// TIA Portal V21 export
FUNCTION_BLOCK "AxisAS_Mng"   // FB81, LAD
TITLE = Positioner + PID / Controllo asse + PID
{ S7_Optimized_Access := 'TRUE' }
VERSION : 1.0
// Positioner with Pid management
// 
// Version from master S7: 2.6
// 
// Date: 2017-08-25
// Project: Mora A.
// 
// Version 2.7: -Corrected maximum speed reached in proportional calculation check.
// Version 2.8: -Used Type for CFG data.
// Gestore ASSE per motore asincrono con posizionatore a generazione di profilo ed inseguimento proporzionale + piramidale
// 
// Michele Montanari
// 
// ver 0.0
// - Curva Trapezio
// - Curva "esse" logaritmica
// - Auto gestione curva per piccoli spostamenti
// - Attesa segnale inverter magnetizzato
// 
// ver 1.0 24/01/2023
// - Curva "esse" Coseno
// - Aggiornamneto struttura
// - Calcolo di tutte le curve in simultanea
// - Arresto #Out in posizione su finestra Vir (da provare.... anche su velocità  == 0)
// - Autogestione (selezione) calcolo acc e dec su definizione prestazioni massime
// - Autogestione (selezione) calcolo velocità possibile in funzione del nuovo target
// - Richiesta abilitazione inverter sempre attiva per abbattere tempo di magentizzazione
// - Inversione al volo del moto
// - Gestione interna del freno motore
// stored: MemoryReserve 100, SetENOAutomatically false
   VAR RETAIN
      DataIn : Struct   // Comando asse
         ixEnablePos { S7_SetPoint := 'True'} : Bool;   // Enable positioner / Abilita asse
         ixDriveReady { S7_SetPoint := 'True'} : Bool;   // Inverter magnetizzato
         ixEnableLevRes { S7_SetPoint := 'True'} : Bool;   // Enable level research / Abilita ricerca livello
         ixAlarmReset { S7_SetPoint := 'True'} : Bool;   // Reset alarms / Reset allarmi
         ixAbort { S7_SetPoint := 'True'} : Bool;   // Initializing motor encoder position / Abort sistema
         ixJogPos { S7_SetPoint := 'True'} : Bool;   // Manual Jog positive / Manuale JOG +
         ixJogNeg { S7_SetPoint := 'True'} : Bool;   // Manual Jog negative / Manuale JOG -
         xAutoSpeedDetect { S7_SetPoint := 'True'} : Bool;   // Calcolo velocità automatico su movimento
         xAutoAccDecCalculation { S7_SetPoint := 'True'} : Bool;   // Calcolo Acc Dec automatico su velocità
         ifPositionRequest { S7_SetPoint := 'True'} : Real;   // Position requested (mm) / Quota richiesta (mm)
         ifSpeedRequest { S7_SetPoint := 'True'} : Real;   // Speed requested (mm/sec) / Velocità richiesta (mm/sec)
         ifPositionStartLev { S7_SetPoint := 'True'} : Real;   // Position start research (mm) / Quota inizio ricerca (mm)
         ifSpeedLev { S7_SetPoint := 'True'} : Real;   // Research speed (mm/sec) / Velocità ricerca (mm/sec)
         ifAccRamp { S7_SetPoint := 'True'} : Real;   // Acceleration ramp (mm/sec^2) / * Rampa accelerazione (mm/sec^2)
         ifDecRamp { S7_SetPoint := 'True'} : Real;   // Deceleration ramp (mm/sec^2) / * Rampa decelerazione (mm/sec^2)
         ifTimeScan { S7_SetPoint := 'True'} : Real;   // Time last scan (sec) / Tempo ultima scansione (sec)
         ifEncoder { S7_SetPoint := 'True'} : Real;   // Actual encoder position (encoder) / Posizione attuale encoder
      END_STRUCT;
      DataOut : Struct   // Gestione Inverte e posizioni
         oxCmdMotorForw : Bool;   // Inverter run enabled / Abilitazione marcia Avanti
         oxCmdMotorBack : Bool;   // Abilitazione marcia Indietro
         oxCmdBrake : Bool;   // Enable brake release / Comando stacco freno
         oxPosError { S7_SetPoint := 'True'} : Bool;   // Pursuit error / Allarme: Errore di inseguimento
         oxEndPos : Bool;   // Positioning terminated / Posizionamento terminato
         oxEndPosBig : Bool;   // Posizionamento Allargato terminato
         oxStopSpeed : Bool;   // Motor speed below low limit / Velocità motore = 0
         oxAccOnWork : Bool;   // Rampa Acc in atto
         oxDecOnWork : Bool;   // Rampa Dec in atto
         ofSpeedRequest : Real;   // Motor speed requested (mm/sec) / Velocita motore richiesta (mm/sec)
         ofEncMotorPos : Real;   // Motor encoder position (mm) / Posizione encoder motore (mm)
         ofMaxError : Real;   // Pursuit max error (mm) / Errore massimo di inseguimento (mm)
         ofSpaceStop : Real;   // Stop space requested from current position/speed (mm) / Spazio richiesto per fermata da posizione/velocità attuale (mm)
         ofSpaceLevRes : Real;   // Spazio richiesto per cambio velocità ricerca livello da posizione/velocità attuale (mm)
         ofSpaceStart : Real;   // Spazio richiesto per partenza da posizione/velocità attuale (mm)
         otTimeMove : Time;   // Tempo ultimo movimento
      END_STRUCT;
      Cfg { S7_SetPoint := 'True'} : "AxixAS_CFG_Type";   // Block data initialisation / Configurazione Asse
      Work : Struct   // Positioner management / Gestione Asse
         xEnablePos { S7_SetPoint := 'True'} : Bool;   // Positioner enabled / Posizionatore abilitato/Positioner enabled
         xINEnable : Bool;   // Memo Posizionatore abilitato per inversione
         xDriveReady { S7_SetPoint := 'True'} : Bool;   // Inverter magnetizzato
         xCmdVirSpeedChanged { S7_SetPoint := 'True'} : Bool;   // Variazione target VEL durante missione
         "xCurveS-L" { S7_SetPoint := 'True'} : Bool;   // Curva non lineare
         "xAutoChangeS-L" { S7_SetPoint := 'True'} : Bool;   // Autoimpostazione LIN per brevi spostamenti
         "xCTRAutoChangeS-L" { S7_SetPoint := 'True'} : Bool;   // Autoimpostazione LIN per brevi spostamenti
         xDecStop { S7_SetPoint := 'True'} : Bool;   // Start dec. for reached requested position / Inizio dec. per raggiungimento quota richiesta
         xDecResearch { S7_SetPoint := 'True'} : Bool;   // Deceleration start for moving to level search speed / Inizio decelerazione per passaggio a velocità ricerca livello
         xStopVirPositioner { S7_SetPoint := 'True'} : Bool;   // Stop positioner for pos. reached / Arresto posizionatore Target raggiunto
         xEnableJog { S7_SetPoint := 'True'} : Bool;   // Jog movement in progress / JOG movimento in corso
         f_PositionTarget { S7_SetPoint := 'True'} : Real;   // Posizione Richiesta Target
         fVirPos { S7_SetPoint := 'True'} : Real;   // Pos. virtual encoder positioner (mm) / Posizione encoder Asse virtuale (mm)
         f_SpeedReqCalc { S7_SetPoint := 'True'} : Real;   // Velocità TARGET autocalcolata su spazio destinazione
         fVirSpeed { S7_SetPoint := 'True'} : Real;   // Virtual encoder speed positioner (mm/sec) / Velocità Asse virtuale (mm/sec) TRA-LOG-COS
         fVirSpeedLinear { S7_SetPoint := 'True'} : Real;   // Velocità Asse LINEARE
         fVirSpeedLog { S7_SetPoint := 'True'} : Real;   // Velocità Asse LOGARITMICA
         fVirSpeedCos { S7_SetPoint := 'True'} : Real;   // Velocità Asse COSENO
         fCmdVirSpeed { S7_SetPoint := 'True'} : Real;   // Virtual encoder current sp(mm/sec) / Velocità richiesta Asse (mm/sec)
         fCmdVirSpeedMemo { S7_SetPoint := 'True'} : Real;   // Memo Velocità richiesta Asse (mm/sec)
         fCmdVirAcc { S7_SetPoint := 'True'} : Real;   // Acc requested for positioner (mm/sec^2) / Acc. richiesta Asse (mm/sec^2)
         fCmdVirDec { S7_SetPoint := 'True'} : Real;   // Dec. requested for positioner (mm/sec^2) / Dec. richiesta Asse (mm/sec^2)
         fLimVirDec { S7_SetPoint := 'True'} : Real;   // Max modulated dec. limit to stop / * Limite massimo dec. modulata per fermata
         fDecVirStop { S7_SetPoint := 'True'} : Real;   // Dec. requested for positioner stop height (mm/sec^2) / * Dec. richiesta per posizionatore stop quota (mm/sec^2)
         fCalcEncErr { S7_SetPoint := 'True'} : Real;   // Error between motor encoder current & real pos. (mm) / * Errore tra pos. attuale e reale encoder motore
         fJogSpeed { S7_SetPoint := 'True'} : Real;   // Speed gen. by jog movement (mm/sec) / Velocità JOG (mm/sec)
         fCmdJogSpeed { S7_SetPoint := 'True'} : Real;   // Speed request to jog movement (mm/sec) / Velocità richiesta JOG (mm/sec)
         fCmdJogAcc { S7_SetPoint := 'True'} : Real;   // Acc. requested for jog movement (mm/sec^2) / Acc. richiesta JOG (mm/sec^2)
         fCmdJogDec { S7_SetPoint := 'True'} : Real;   // Dec. requested for jog movement (mm/sec^2) / Dec. richiesta JOG (mm/sec^2)
         "fLim+Ppid" { S7_SetPoint := 'True'} : Real;   // Proportional action positive maximum limit (1/5 max speed) / Limite massimo positivo azione proporzionale (20% velocità massima)
         "fLim-Ppid" { S7_SetPoint := 'True'} : Real;   // Proportional action negative maximum limit (1/5 max speed) / Limite massimo negativo azione proporzionale (20% velocità massima)
         fCmdSpeedMot { S7_SetPoint := 'True'} : Real;   // Motor control speed from positioner o Jog / Velocità comando motore da POS o JOG
         fSuppCalcPpid { S7_SetPoint := 'True'} : Real;   // Proportional calculation supp. / App calcolo proporzionale
         fMemoMaxSpeed { S7_SetPoint := 'True'} : Real;   // Store maximum speed (mm/sec) / Memorizzo velocità massima (mm/sec)
         fPpid { S7_SetPoint := 'True'} : Real;   // Part P of Pid / Parte P del Pid
         fMemoOldPos { S7_SetPoint := 'True'} : Real;   // Quota Old/Position Old (mm)
         fAccOnWork { S7_SetPoint := 'True'} : Real;   // Accelerazione calcolata/imposta
         fDecOnWork { S7_SetPoint := 'True'} : Real;   // Decelerazione calcolata/imposta
         xTimBrakeDelay_Fwd : Bool;   // Ritardo sgancio freno FWD
         xTimBrakeDelay_Bkw : Bool;   // Ritardo sgancio freno BKW
         xTimStopEndPos : Bool;   // Ritardo allarme controllo fine posizionamento
         fCalc : Array[0..20] of Real;
         xCalc : Array[0..20] of Bool;
      END_STRUCT;
   END_VAR
   VAR
      TmrBrake_Fwd : IEC_TIMER;   // Timer sgancio freno FWD
      TmrBrake_Bkw : IEC_TIMER;   // Timer sgancio freno BKW
      Tmr_EndPos : IEC_TIMER;   // Timer allarme controllo fine posizionamento
      Tmr_DriveOnReq : IEC_TIMER;   // Timer OFF richiesta Drive Ready
      Tmr_OnMove : IEC_TIMER;
   END_VAR
   VAR_TEMP
      tfSuppCalc : Real;   // Calculation support / Appoggio per calcoli
      fSlopeAccLog : Real;
      fSlopeDecLog : Real;
      fSlopeAccCos : Real;
      fSlopeDecCos : Real;
      fCalcSpeed : Real;
      oxCmdMotorFWD : Bool;
      oxCmdMotorBKW : Bool;
      fCalcSpaceOff : Real;
      xDummy : Bool;
   END_VAR
   VAR CONSTANT
      PiGrego : Real := 3.141593;
      "100Sec" : Time := T#100s;
   END_VAR
   VAR_TEMP   // added for the SCL form of the ladder/FBD networks
      _w1 : Bool;
      _w2 : Bool;
      _w3 : Bool;
   END_VAR
BEGIN

REGION Network 1 (SCL): Autocalcolo velocità su spazio da percorrere
   IF #DataIn.xAutoSpeedDetect THEN
       IF #Cfg."xmm/degree" THEN
           IF ABS(#DataIn.ifPositionRequest - #DataIn.ifEncoder) >= #Cfg.fMaxSpeed / 2 THEN
               #Work.f_SpeedReqCalc := #DataIn.ifSpeedRequest;
           ELSE
               #fCalcSpeed := ABS(#DataIn.ifPositionRequest - #DataIn.ifEncoder);
               IF NOT #DataOut.oxCmdMotorForw AND NOT #DataOut.oxCmdMotorBack THEN
                   IF #fCalcSpeed <= #DataIn.ifSpeedRequest THEN
                       #Work.f_SpeedReqCalc := #fCalcSpeed;
                   ELSE
                       #Work.f_SpeedReqCalc := #DataIn.ifSpeedRequest;
                   END_IF;
               END_IF;
           END_IF;
       ELSE
           IF ABS(#DataIn.ifPositionRequest - #DataIn.ifEncoder) >= 60.0 THEN
               #Work.f_SpeedReqCalc := #DataIn.ifSpeedRequest;
           ELSE
               #fCalcSpeed := ABS(#DataIn.ifPositionRequest - #DataIn.ifEncoder);
               IF NOT #DataOut.oxCmdMotorForw AND NOT #DataOut.oxCmdMotorBack THEN
                   IF #fCalcSpeed <= #DataIn.ifSpeedRequest THEN
                       #Work.f_SpeedReqCalc := #fCalcSpeed;
                   ELSE
                       #Work.f_SpeedReqCalc := #DataIn.ifSpeedRequest;
                   END_IF;
               END_IF;
           END_IF;
       END_IF;
   ELSE
       #Work.f_SpeedReqCalc := #DataIn.ifSpeedRequest;
   END_IF;

   IF #Work.f_SpeedReqCalc > #Cfg.fMaxSpeed THEN
       #Work.f_SpeedReqCalc := #Cfg.fMaxSpeed;
   END_IF;
END_REGION

REGION Network 2: Memo Posizionatore abilitato per inversione
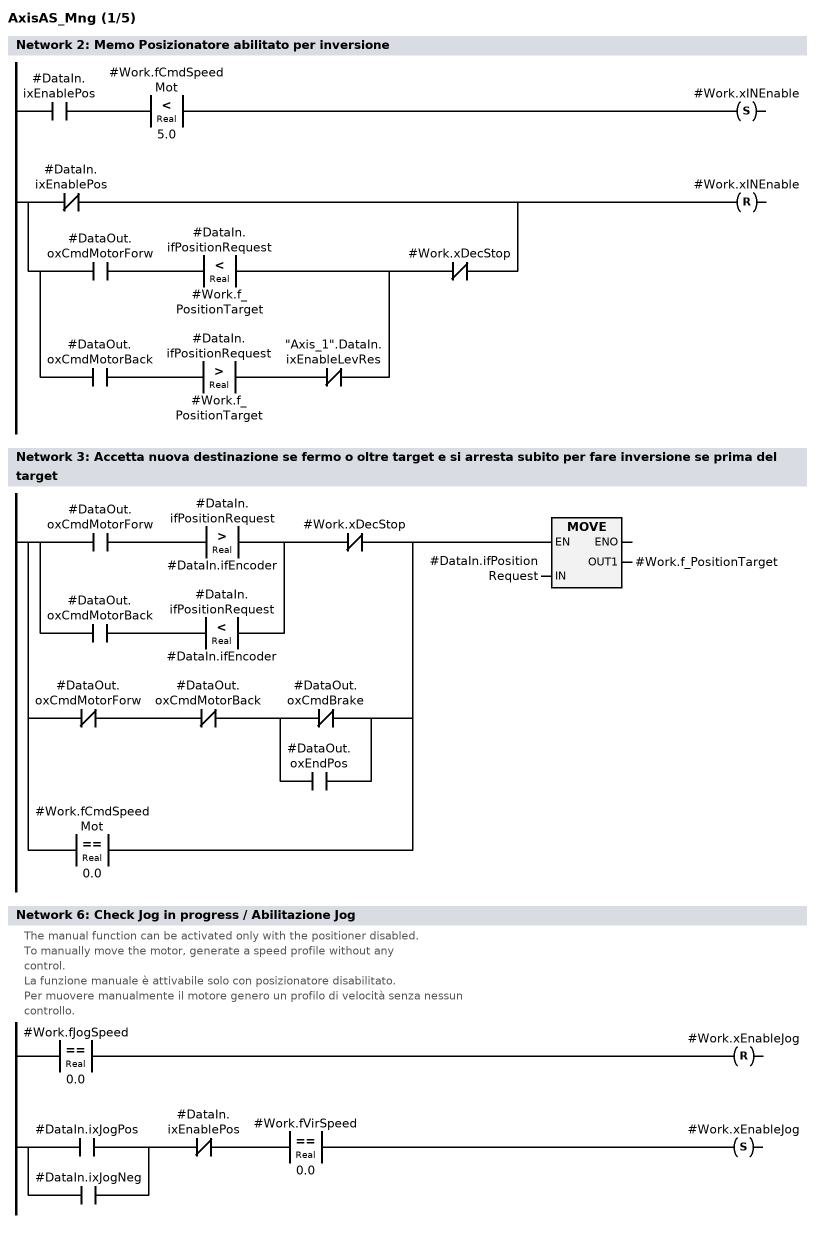
   RUNG wire#powerrail
      Contact( #DataIn.ixEnablePos )
      { S7_Templates := "SrcType := Real" } LT_Contact(in1 := #Work.fCmdSpeedMot, in2 := 5.0)
      S_Coil( #Work.xINEnable )
   END_RUNG
   RUNG wire#powerrail
      I_Contact( #DataIn.ixEnablePos )
      wire#w1
      R_Coil( #Work.xINEnable )
   END_RUNG
   RUNG wire#powerrail
      Contact( #DataOut.oxCmdMotorForw )
      { S7_Templates := "SrcType := Real" } LT_Contact(in1 := #DataIn.ifPositionRequest, in2 := #Work.f_PositionTarget)
      wire#w2
      I_Contact( #Work.xDecStop )
   END_RUNG wire#w1
   RUNG wire#powerrail
      Contact( #DataOut.oxCmdMotorBack )
      { S7_Templates := "SrcType := Real" } GT_Contact(in1 := #DataIn.ifPositionRequest, in2 := #Work.f_PositionTarget)
      I_Contact( "Axis_1".DataIn.ixEnableLevRes )
   END_RUNG wire#w2
   // the same network as SCL:
   IF #DataIn.ixEnablePos AND (#Work.fCmdSpeedMot < 5.0) THEN #Work.xINEnable := TRUE; END_IF;
   IF NOT #DataIn.ixEnablePos OR (((#DataOut.oxCmdMotorForw AND (#DataIn.ifPositionRequest < #Work.f_PositionTarget)) OR (#DataOut.oxCmdMotorBack AND (#DataIn.ifPositionRequest > #Work.f_PositionTarget) AND NOT "Axis_1".DataIn.ixEnableLevRes)) AND NOT #Work.xDecStop) THEN
       #Work.xINEnable := FALSE;
   END_IF;
END_REGION

REGION Network 3: Accetta nuova destinazione se fermo o oltre target e si arresta subito per fare inversione se prima del target
   RUNG wire#powerrail
      Contact( #DataOut.oxCmdMotorForw )
      { S7_Templates := "SrcType := Real" } GT_Contact(in1 := #DataIn.ifPositionRequest, in2 := #DataIn.ifEncoder)
      wire#w1
      I_Contact( #Work.xDecStop )
      wire#w2
      Move(in := #DataIn.ifPositionRequest, out1 => #Work.f_PositionTarget)
   END_RUNG
   RUNG wire#powerrail
      Contact( #DataOut.oxCmdMotorBack )
      { S7_Templates := "SrcType := Real" } LT_Contact(in1 := #DataIn.ifPositionRequest, in2 := #DataIn.ifEncoder)
   END_RUNG wire#w1
   RUNG wire#powerrail
      I_Contact( #DataOut.oxCmdMotorForw )
      I_Contact( #DataOut.oxCmdMotorBack )
      wire#w3
      I_Contact( #DataOut.oxCmdBrake )
   END_RUNG wire#w2
   RUNG wire#w3
      Contact( #DataOut.oxEndPos )
   END_RUNG wire#w2
   RUNG wire#powerrail
      { S7_Templates := "SrcType := Real" } EQ_Contact(in1 := #Work.fCmdSpeedMot, in2 := 0.0)
   END_RUNG wire#w2
   // the same network as SCL:
   IF (((#DataOut.oxCmdMotorForw AND (#DataIn.ifPositionRequest > #DataIn.ifEncoder)) OR (#DataOut.oxCmdMotorBack AND (#DataIn.ifPositionRequest < #DataIn.ifEncoder))) AND NOT #Work.xDecStop) OR (NOT #DataOut.oxCmdMotorForw AND NOT #DataOut.oxCmdMotorBack AND (NOT #DataOut.oxCmdBrake OR #DataOut.oxEndPos)) OR (#Work.fCmdSpeedMot = 0.0) THEN
       #Work.f_PositionTarget := #DataIn.ifPositionRequest;
   END_IF;
END_REGION

REGION Network 4 (SCL): Autocalcolo ACC-DEC su velocità
   IF #DataIn.xAutoAccDecCalculation THEN

       #Work.fAccOnWork := #Cfg.fMaxAccRamp * (#Work.f_SpeedReqCalc / #Cfg.fMaxSpeed);
       #Work.fDecOnWork := #Cfg.fMaxDecRamp * (#Work.f_SpeedReqCalc / #Cfg.fMaxSpeed);

       IF #Cfg."xmm/degree" THEN
           IF #Work.fAccOnWork < 100 THEN
               #Work.fAccOnWork := 100;
           END_IF;
           IF #Work.fDecOnWork < 100 THEN
               #Work.fDecOnWork := 100;
           END_IF;
       ELSE
           IF #Work.fAccOnWork < 20 THEN
               #Work.fAccOnWork := 20;
           END_IF;
           IF #Work.fDecOnWork < 20 THEN
               #Work.fDecOnWork := 20;
           END_IF;
       END_IF;

   ELSE

       #Work.fAccOnWork := #DataIn.ifAccRamp;
       #Work.fDecOnWork := #DataIn.ifDecRamp;

   END_IF;
END_REGION

REGION Network 5 (SCL): Encoder value conversion / Selezione curva
   // Per spostamenti inferiori a  #CFG."fAutoChangeS-Lvalue" impone una curva a TRA se selezionata LOG
   IF #Cfg."xCurveS-L" = 0 THEN
       #Work."xCurveS-L" := FALSE;
   END_IF;

   IF #Cfg."xCurveS-L" = 1 THEN
       IF (#Work.xINEnable) AND NOT #Work."xCTRAutoChangeS-L" THEN
           #Work."xCTRAutoChangeS-L" := TRUE;
           IF (ABS(#Work.f_PositionTarget - #DataOut.ofEncMotorPos) < #Cfg."fAutoChangeS-Lvalue") THEN
               #Work."xAutoChangeS-L" := TRUE;
           END_IF;
       END_IF;
       IF #Work."xAutoChangeS-L" THEN
           #Work."xCurveS-L" := FALSE;
       ELSE
           #Work."xCurveS-L" := TRUE;
       END_IF;
   END_IF;

   IF #Cfg."xCurveS-L" = 2 THEN
       #Work."xCurveS-L" := TRUE;
   END_IF;

   IF NOT #Work.xINEnable AND NOT #Work.xDecStop THEN
       #Work."xCTRAutoChangeS-L" := FALSE;
   END_IF;

   IF ABS(#Work.f_PositionTarget - #DataOut.ofEncMotorPos) <= #Cfg.fVirt_EncWindPos THEN
       #Work."xAutoChangeS-L" := FALSE;

   END_IF;
END_REGION

REGION Network 6: Check Jog in progress / Abilitazione Jog
   // The manual function can be activated only with the positioner disabled.
   // To manually move the motor, generate a speed profile without any 
   // control.
   // La funzione manuale è attivabile solo con posizionatore disabilitato.
   // Per muovere manualmente il motore genero un profilo di velocità senza nessun 
   // controllo.
   RUNG wire#powerrail
      { S7_Templates := "SrcType := Real" } EQ_Contact(in1 := #Work.fJogSpeed, in2 := 0.0)
      R_Coil( #Work.xEnableJog )
   END_RUNG
   RUNG wire#powerrail
      Contact( #DataIn.ixJogPos )
      wire#w1
      I_Contact( #DataIn.ixEnablePos )
      { S7_Templates := "SrcType := Real" } EQ_Contact(in1 := #Work.fVirSpeed, in2 := 0.0)
      S_Coil( #Work.xEnableJog )
   END_RUNG
   RUNG wire#powerrail
      Contact( #DataIn.ixJogNeg )
   END_RUNG wire#w1
   // the same network as SCL:
   IF #Work.fJogSpeed = 0.0 THEN #Work.xEnableJog := FALSE; END_IF;
   IF (#DataIn.ixJogPos OR #DataIn.ixJogNeg) AND NOT #DataIn.ixEnablePos AND (#Work.fVirSpeed = 0.0) THEN
       #Work.xEnableJog := TRUE;
   END_IF;
END_REGION

REGION Network 7 (SCL): Jog operation activation / Attivazione funzionamento di jog
   // Con abilitazione attiva carico velocità jog e inizio generazione profilo di velocità senza alcun controllo
   IF #Work.xEnableJog THEN

       IF #DataIn.ixJogPos OR #DataIn.ixJogNeg THEN
           #Work.fCmdJogSpeed := #Cfg.fJogSpeed;
       ELSE
           #Work.fCmdJogSpeed := 0.0;
       END_IF;

       IF #Work.fJogSpeed >= 0.0 THEN
           #Work.fCmdJogAcc := #Cfg.fJogAcc * #DataIn.ifTimeScan;
           #Work.fCmdJogDec := #Cfg.fJogDec * #DataIn.ifTimeScan;
       END_IF;

       IF #Work.fCmdJogSpeed > #Work.fJogSpeed THEN
           #Work.fJogSpeed := #Work.fJogSpeed + #Work.fCmdJogAcc;
           IF #Work.fJogSpeed > #Work.fCmdJogSpeed THEN
               #Work.fJogSpeed := #Work.fCmdJogSpeed;
           END_IF;
       END_IF;

       IF #Work.fCmdJogSpeed < #Work.fJogSpeed THEN
           #Work.fJogSpeed := #Work.fJogSpeed - #Work.fCmdJogDec;
           IF #Work.fJogSpeed < #Work.fCmdJogSpeed THEN
               #Work.fJogSpeed := #Work.fCmdJogSpeed;
           END_IF;
       END_IF;

   END_IF;
END_REGION

REGION Network 8: Check if positioner is enabled / Controllo se posizionatore abilitato e inverter ready
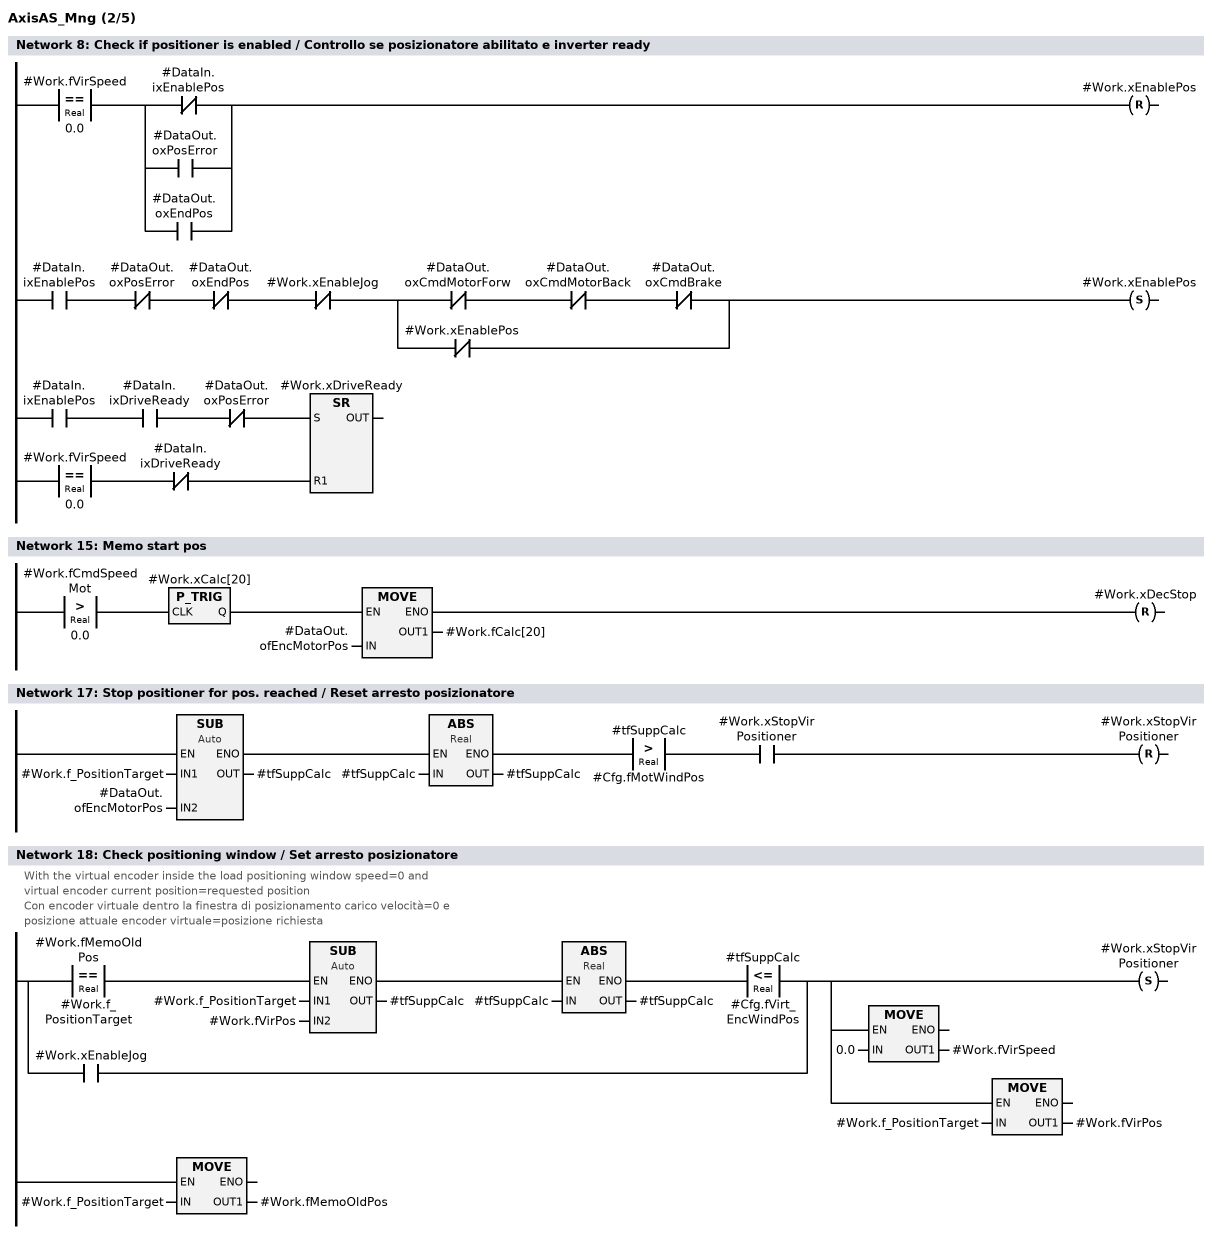
   RUNG wire#powerrail
      { S7_Templates := "SrcType := Real" } EQ_Contact(in1 := #Work.fVirSpeed, in2 := 0.0)
      wire#w1
      I_Contact( #DataIn.ixEnablePos )
      wire#w2
      R_Coil( #Work.xEnablePos )
   END_RUNG
   RUNG wire#w1
      Contact( #DataOut.oxPosError )
   END_RUNG wire#w2
   RUNG wire#w1
      Contact( #DataOut.oxEndPos )
   END_RUNG wire#w2
   RUNG wire#powerrail
      Contact( #DataIn.ixEnablePos )
      I_Contact( #DataOut.oxPosError )
      I_Contact( #DataOut.oxEndPos )
      I_Contact( #Work.xEnableJog )
      wire#w3
      I_Contact( #DataOut.oxCmdMotorForw )
      I_Contact( #DataOut.oxCmdMotorBack )
      I_Contact( #DataOut.oxCmdBrake )
      wire#w4
      S_Coil( #Work.xEnablePos )
   END_RUNG
   RUNG wire#w3
      I_Contact( #Work.xEnablePos )
   END_RUNG wire#w4
   RUNG wire#powerrail
      Contact( #DataIn.ixEnablePos )
      Contact( #DataIn.ixDriveReady )
      I_Contact( #DataOut.oxPosError )
      S_SR(operand := #Work.xDriveReady, r1 := wire#w5)
   END_RUNG
   RUNG wire#powerrail
      { S7_Templates := "SrcType := Real" } EQ_Contact(in1 := #Work.fVirSpeed, in2 := 0.0)
      I_Contact( #DataIn.ixDriveReady )
   END_RUNG wire#w5
   // the same network as SCL:
   IF (#Work.fVirSpeed = 0.0) AND (NOT #DataIn.ixEnablePos OR #DataOut.oxPosError OR #DataOut.oxEndPos) THEN
       #Work.xEnablePos := FALSE;
   END_IF;
   IF #DataIn.ixEnablePos AND NOT #DataOut.oxPosError AND NOT #DataOut.oxEndPos AND NOT #Work.xEnableJog AND ((NOT #DataOut.oxCmdMotorForw AND NOT #DataOut.oxCmdMotorBack AND NOT #DataOut.oxCmdBrake) OR NOT #Work.xEnablePos) THEN
       #Work.xEnablePos := TRUE;
   END_IF;
   IF #DataIn.ixEnablePos AND #DataIn.ixDriveReady AND NOT #DataOut.oxPosError THEN
       #Work.xDriveReady := TRUE;   // SR flip-flop
   END_IF;
   IF (#Work.fVirSpeed = 0.0) AND NOT #DataIn.ixDriveReady THEN #Work.xDriveReady := FALSE; END_IF;
END_REGION

REGION Network 9 (SCL): Calcolo Profilo velocità posizionatore TRAPEZIO

   #Work.fCmdVirAcc := (#Work.fAccOnWork * #DataIn.ifTimeScan);
   #Work.fCmdVirDec := (#Work.fDecOnWork * #DataIn.ifTimeScan);

   IF #Work.fCmdVirSpeed > #Work.fVirSpeedLinear THEN
       #Work.fVirSpeedLinear := #Work.fVirSpeedLinear + #Work.fCmdVirAcc;
       IF #Work.fVirSpeedLinear > #Work.fCmdVirSpeed THEN
           #Work.fVirSpeedLinear := #Work.fCmdVirSpeed;
       END_IF;
   END_IF;

   IF #Work.fCmdVirSpeed <= #Work.fVirSpeedLinear THEN
       #Work.fVirSpeedLinear := #Work.fVirSpeedLinear - #Work.fCmdVirDec;
       IF #Work.fVirSpeedLinear < #Work.fCmdVirSpeed THEN
           #Work.fVirSpeedLinear := #Work.fCmdVirSpeed;
       END_IF;
       IF NOT (#Work.xStopVirPositioner) AND (#Work.fVirSpeedLinear < #Cfg.fMinSpeed)
           AND NOT (#DataOut.oxPosError) AND #Work.xINEnable AND #Work.xDriveReady THEN
           #Work.fVirSpeedLinear := #Cfg.fMinSpeed;
       END_IF;
   END_IF;
END_REGION

REGION Network 10 (SCL): Gestione cambio target velocità LOG-COS
       IF (#Work.fCmdVirSpeedMemo <> #Work.fCmdVirSpeed) THEN
           IF #Work.fCmdVirSpeed > 0 AND #Work.fCmdVirSpeedMemo <> 0 THEN
               #Work.fCalc[7] := #Work.fVirSpeedLog;
               #Work.fCalc[0] := 0;
               #Work.fCalc[17] := #Work.fVirSpeedCos;
               #Work.fCalc[19] := 0;
               IF #Work.fCmdVirSpeed > #Work.fCmdVirSpeedMemo THEN
                   #Work.xCmdVirSpeedChanged := FALSE;
               ELSE
                   #Work.xCmdVirSpeedChanged := TRUE;
               END_IF;
           END_IF;
           #Work.fCmdVirSpeedMemo := #Work.fCmdVirSpeed;
       END_IF;
END_REGION

REGION Network 11 (SCL): Calculate positioner speed / Calcolo Profilo velocità posizionatore Logaritmica
   // Calculate speed positioner profile.
   // During the stop phase, module the deceleration to stop in the position 
   // requested; the maximum deceleration variation is 50%. This is 
   // necessary because the 0 speed request point is afflicted by an error 
   // generated by the CPU scanning time.
   // Calcolo velocità profilo posizionatore.
   // Durante la fase di fermata modulo la decelerazione per fermarmi nella posizione 
   // richiesta; la variazione massima di decelerazione è del 50%. Questo è 
   // necessario in quanto il punto di richiesta velocità 0 è afflitto dall'errore 
   // generato dal tempo di scansione della CPU.

   IF #Work."xCurveS-L" THEN



       IF  #Work.fCalc[10] < #Work.fVirSpeedLog THEN
           #Work.fCalc[10] := #Work.fVirSpeedLog;
       END_IF;
       IF #Work.fVirSpeed = 0 THEN
           #Work.fCalc[10] := 0;
       END_IF;


       #fSlopeAccLog := (12 * #Work.fAccOnWork) / (ABS(#Work.fCmdVirSpeed - #Work.fCalc[7]) + 1);
       #fSlopeDecLog := (12 * #Work.fDecOnWork) / (#Work.fCalc[10] + 1);


       IF #Work.fCmdVirSpeed > 0 THEN

           #Work.fCalc[5] := 1;
           IF #Work.fCalc[5] < #Work.fVirSpeedLog THEN
               #Work.fCalc[5] := #Work.fVirSpeedLog;
           END_IF;
           #Work.fCalc[0] := #Work.fCalc[0] + #DataIn.ifTimeScan;
           IF NOT #Work.xCmdVirSpeedChanged THEN
               #Work.fVirSpeedLog := #Work.fCalc[7] + (#Work.fCmdVirSpeed - #Work.fCalc[7]) * (1 / (1 + EXP(- (#Work.fCalc[0] * #fSlopeAccLog - #Cfg.fFirstStepNepero))));
           ELSE
               #fSlopeDecLog := (12 * #Work.fDecOnWork) / ABS((#Work.fCalc[7] - #Work.fCmdVirSpeed) + 1);
               #Work.fVirSpeedLog := #Work.fCalc[7] + (#Work.fCmdVirSpeed - #Work.fCalc[7]) * (1 / (1 + EXP(- (#Work.fCalc[0] * #fSlopeDecLog - #Cfg.fFirstStepNepero))));
           END_IF;

           #Work.fCalc[4] := 0;


       ELSE

           IF #Work.fVirSpeedLog > 0 THEN
               #Work.fCalc[4] := #Work.fCalc[4] + #DataIn.ifTimeScan;
           END_IF;
           #fSlopeDecLog := (12 * #Work.fDecOnWork) / (#Work.fCalc[5] + 1);
           #Work.fVirSpeedLog := #Work.fCalc[5] * (1 - (1 / (1 + EXP(- ((#Work.fCalc[4]) * #fSlopeDecLog - #Cfg.fFirstStepNepero)))));
           #Work.fCalc[10] := #Work.fCalc[5];
           #Work.fCalc[7] := #Work.fVirSpeedLog;
           #Work.fCalc[0] := 0;
       END_IF;


       IF #Work.xStopVirPositioner THEN
               #Work.fVirSpeed := 0;
               #Work.fCalc[0] := 0;
               #Work.fCalc[4] := 0;
               #Work.fCalc[5] := 0;
               #Work.fCalc[7] := 0;
        END_IF;

   END_IF;
END_REGION

REGION Network 12 (SCL): Calculate positioner speed / Calcolo Profilo velocità posizionatore Coseno
   // Calculate speed positioner profile.
   // During the stop phase, module the deceleration to stop in the position 
   // requested; the maximum deceleration variation is 50%. This is 
   // necessary because the 0 speed request point is afflicted by an error 
   // generated by the CPU scanning time.
   // Calcolo velocità profilo posizionatore.
   // Durante la fase di fermata modulo la decelerazione per fermarmi nella posizione 
   // richiesta; la variazione massima di decelerazione è del 50%. Questo è 
   // necessario in quanto il punto di richiesta velocità 0 è afflitto dall'errore 
   // generato dal tempo di scansione della CPU.

   IF #Work."xCurveS-L" THEN


       IF #Work.fCmdVirSpeed > 0 THEN

           #Work.fCalc[19] := #Work.fCalc[19] + #DataIn.ifTimeScan;

                   #Work.fCalc[13] := 1;
                   IF #Work.fCalc[13] < #Work.fVirSpeedCos THEN
                       #Work.fCalc[13] := #Work.fVirSpeedCos;
                   END_IF;
                   #fSlopeAccCos := #PiGrego / ((ABS(#Work.fCmdVirSpeed - #Work.fCalc[17]) + 1) / #Work.fAccOnWork);
                   IF NOT #Work.xCmdVirSpeedChanged THEN
                       IF #fSlopeAccCos * #Work.fCalc[19] < #PiGrego THEN
                           #Work.fVirSpeedCos := #Work.fCalc[17] + (#Work.fCmdVirSpeed - #Work.fCalc[17]) * 0.5 * (COS(#fSlopeAccCos * #Work.fCalc[19] + #PiGrego) + 1);
                       ELSE
                           #Work.fVirSpeedCos := #Work.fCmdVirSpeed;
                       END_IF;
                   ELSE
                       #fSlopeDecCos := #PiGrego / ((ABS(#Work.fCmdVirSpeed - #Work.fCalc[17]) + 1) / #Work.fDecOnWork);
                       IF #fSlopeDecCos * #Work.fCalc[19] < #PiGrego THEN
                           #Work.fVirSpeedCos := #Work.fCalc[17] + (#Work.fCmdVirSpeed - #Work.fCalc[17]) * 0.5 * (COS(#fSlopeDecCos * #Work.fCalc[19] + #PiGrego) + 1);
                       ELSE
                           #Work.fVirSpeedCos := #Work.fCmdVirSpeed;
                       END_IF;

                   END_IF;
               #Work.fCalc[18] := #DataIn.ifTimeScan * 0;

           ELSE
               #Work.fCalc[19] := 0;
               IF #Work.fVirSpeedCos > 0 THEN
                   #Work.fCalc[18] := #Work.fCalc[18] + #DataIn.ifTimeScan;
                   #fSlopeDecCos := #PiGrego / (#Work.fCalc[13] / #Work.fDecOnWork);
                   IF #fSlopeDecCos * #Work.fCalc[18] < #PiGrego THEN
                       #Work.fVirSpeedCos := #Work.fCalc[13] * 0.5 * (COS(#fSlopeDecCos * #Work.fCalc[18]) + 1);
                   ELSE
                       #Work.fVirSpeedCos := 0;
                   END_IF;
                   #Work.fCalc[17] := #Work.fVirSpeedCos;
                   #Work.fCalc[19] := 0;
               END_IF;


       END_IF;


           IF #Work.xStopVirPositioner THEN
               #Work.fVirSpeed := 0;
               #Work.fCalc[13] := 0;
               #Work.fCalc[17] := 0;
               #Work.fCalc[18] := 0;
               #Work.fCalc[19] := 0;
           END_IF;


   END_IF;
END_REGION

REGION Network 13 (SCL): Gestione profilo posizionatore

   IF NOT #Work.xStopVirPositioner THEN

       CASE #Cfg."xCurveS-L" OF
           0:
               #Work.fVirSpeed := #Work.fVirSpeedLinear;
           1:
               IF #Work."xCurveS-L" THEN
                   IF #Work.fVirSpeedLog >= 1 THEN
                       #Work.fVirSpeed := #Work.fVirSpeedLog;
                   ELSE
                       #Work.fVirSpeed := 0;
                   END_IF;
               ELSE
                   #Work.fVirSpeed := #Work.fVirSpeedLinear;
               END_IF;

           2:
               #Work.fVirSpeed := #Work.fVirSpeedCos;

       END_CASE;


       IF (#Work.fVirSpeed < #Cfg.fMinSpeed) AND #Work.xINEnable AND NOT (#DataOut.oxPosError) AND #Work.xDriveReady THEN
           #Work.fVirSpeed := #Cfg.fMinSpeed;
       END_IF;
   ELSE
       #Work.xCmdVirSpeedChanged := FALSE;
   END_IF;
END_REGION

REGION Network 14 (SCL): Calculate pos. compared to speed / Calcolo posizione con legge di moto
   // Calculate the profile generator position according to speed and time 
   // for scanning of the CPU.
   // The virtual encoder generated in this way is needed to calculate the PID managing the 
   // motor
   // Calcolo la posizione del generatore di profilo sul tempo 
   // di scansione della CPU.
   IF NOT #Work.xStopVirPositioner THEN
       IF #Work.f_PositionTarget > #Work.fVirPos THEN
           #Work.fVirPos := #Work.fVirPos + (#Work.fVirSpeed * #DataIn.ifTimeScan);
       ELSE
           #Work.fVirPos := #Work.fVirPos - (#Work.fVirSpeed * #DataIn.ifTimeScan);
       END_IF;
   END_IF;
END_REGION

REGION Network 15: Memo start pos
   RUNG wire#powerrail
      { S7_Templates := "SrcType := Real" } GT_Contact(in1 := #Work.fCmdSpeedMot, in2 := 0.0)
      P_Trig( #Work.xCalc[20] )
      Move(in := #DataOut.ofEncMotorPos, out1 => #Work.fCalc[20])
      R_Coil( #Work.xDecStop )
   END_RUNG
   // the same network as SCL:
   #_w1 := #Work.fCmdSpeedMot > 0.0;
   #_w2 := #_w1 AND NOT #Work.xCalc[20];   // rising edge
   #Work.xCalc[20] := #_w1;
   IF #_w2 THEN
       #Work.fCalc[20] := #DataOut.ofEncMotorPos;
       #Work.xDecStop := FALSE;
   END_IF;
END_REGION

REGION Network 16 (SCL): Check when it is time to bring the speed to 0 to stop / Calcolo spazio di arresto del profilo con dati attuali
   #DataOut.ofSpaceStop := #Cfg.fMotWindPos + #Cfg.fMotAdvStopPosition + (SQR(#Work.fVirSpeed)) / (#Work.fDecOnWork * 2.0);
   #DataOut.ofSpaceStart := (SQR(#Work.fCmdVirSpeed)) / (#Work.fAccOnWork * 2.0);
   #DataOut.ofSpaceLevRes := (SQR(#Work.fVirSpeed) / (#Work.fDecOnWork * 2.0)) - (SQR( #DataIn.ifSpeedLev) / (#Work.fDecOnWork * 2.0)) + 50;
   // #OUT.ofSpaceLevRes := (SQR(#WORK.f_SpeedReqCalc ) / (#IN.ifDecRamp * 2.0)) - (SQR( #IN.ifSpeedLev) / (#IN.ifDecRamp * 2.0));

   #DataOut.oxAccOnWork := ABS(#Work.fCalc[20] - #DataOut.ofEncMotorPos) < #DataOut.ofSpaceStart;
   #DataOut.oxDecOnWork := #Work.xDecStop OR ((#Work.fCmdSpeedMot > 0) AND NOT #Work.xINEnable);


   IF (ABS(#Work.f_PositionTarget - #Work.fVirPos)) <= #DataOut.ofSpaceStop THEN
       #Work.xDecStop := 1;
   END_IF;

   IF NOT (#Work.xEnablePos) OR #Work.xStopVirPositioner THEN //OR (NOT(#OUT.oxCmdMotorForw) AND NOT(#OUT.oxCmdMotorBack)) THEN
       #Work.xDecStop := 0;
   END_IF;


   IF #DataIn.ixEnableLevRes AND #Work.xINEnable THEN //AND (#SUPPORT.fVirSpeed > 0)   AND  #OUT.oxCmdMotorBack
       IF #DataIn.ifEncoder < (#DataIn.ifPositionStartLev + #DataOut.ofSpaceLevRes + 1) THEN
           #Work.xDecResearch := 1;
       END_IF;
   ELSE
       #Work.xDecResearch := 0;
   END_IF;
END_REGION

REGION Network 17: Stop positioner for pos. reached / Reset arresto posizionatore
   RUNG wire#powerrail
      Sub(in1 := #Work.f_PositionTarget, in2 := #DataOut.ofEncMotorPos, out => #tfSuppCalc)
      { S7_Templates := "SrcType := Real" } Abs(in := #tfSuppCalc, out => #tfSuppCalc)
      { S7_Templates := "SrcType := Real" } GT_Contact(in1 := #tfSuppCalc, in2 := #Cfg.fMotWindPos)
      Contact( #Work.xStopVirPositioner )
      R_Coil( #Work.xStopVirPositioner )
   END_RUNG
   // the same network as SCL:
   #tfSuppCalc := #Work.f_PositionTarget - #DataOut.ofEncMotorPos;
   #tfSuppCalc := ABS(#tfSuppCalc);
   IF (#tfSuppCalc > #Cfg.fMotWindPos) AND #Work.xStopVirPositioner THEN
       #Work.xStopVirPositioner := FALSE;
   END_IF;
END_REGION

REGION Network 18: Check positioning window / Set arresto posizionatore
   // With the virtual encoder inside the load positioning window speed=0 and 
   // virtual encoder current position=requested position
   // Con encoder virtuale dentro la finestra di posizionamento carico velocità=0 e 
   // posizione attuale encoder virtuale=posizione richiesta
   RUNG wire#powerrail
      { S7_Templates := "SrcType := Real" } EQ_Contact(in1 := #Work.fMemoOldPos, in2 := #Work.f_PositionTarget)
      Sub(in1 := #Work.f_PositionTarget, in2 := #Work.fVirPos, out => #tfSuppCalc)
      { S7_Templates := "SrcType := Real" } Abs(in := #tfSuppCalc, out => #tfSuppCalc)
      { S7_Templates := "SrcType := Real" } LE_Contact(in1 := #tfSuppCalc, in2 := #Cfg.fVirt_EncWindPos)
      wire#w1
      S_Coil( #Work.xStopVirPositioner )
   END_RUNG
   RUNG wire#powerrail
      Contact( #Work.xEnableJog )
   END_RUNG wire#w1
   RUNG wire#w1
      Move(in := 0.0, out1 => #Work.fVirSpeed)
   END_RUNG
   RUNG wire#w1
      Move(in := #Work.f_PositionTarget, out1 => #Work.fVirPos)
   END_RUNG
   RUNG wire#powerrail
      Move(in := #Work.f_PositionTarget, out1 => #Work.fMemoOldPos)
   END_RUNG
   // the same network as SCL:
   #_w1 := #Work.fMemoOldPos = #Work.f_PositionTarget;
   IF #_w1 THEN
       #tfSuppCalc := #Work.f_PositionTarget - #Work.fVirPos;
       #tfSuppCalc := ABS(#tfSuppCalc);
   END_IF;
   IF (#_w1 AND (#tfSuppCalc <= #Cfg.fVirt_EncWindPos)) OR #Work.xEnableJog THEN
       #Work.xStopVirPositioner := TRUE;
       #Work.fVirSpeed := 0.0;
       #Work.fVirPos := #Work.f_PositionTarget;
   END_IF;
   #Work.fMemoOldPos := #Work.f_PositionTarget;
END_REGION

REGION Network 19: Positioning speed requested / Velocità richiesta
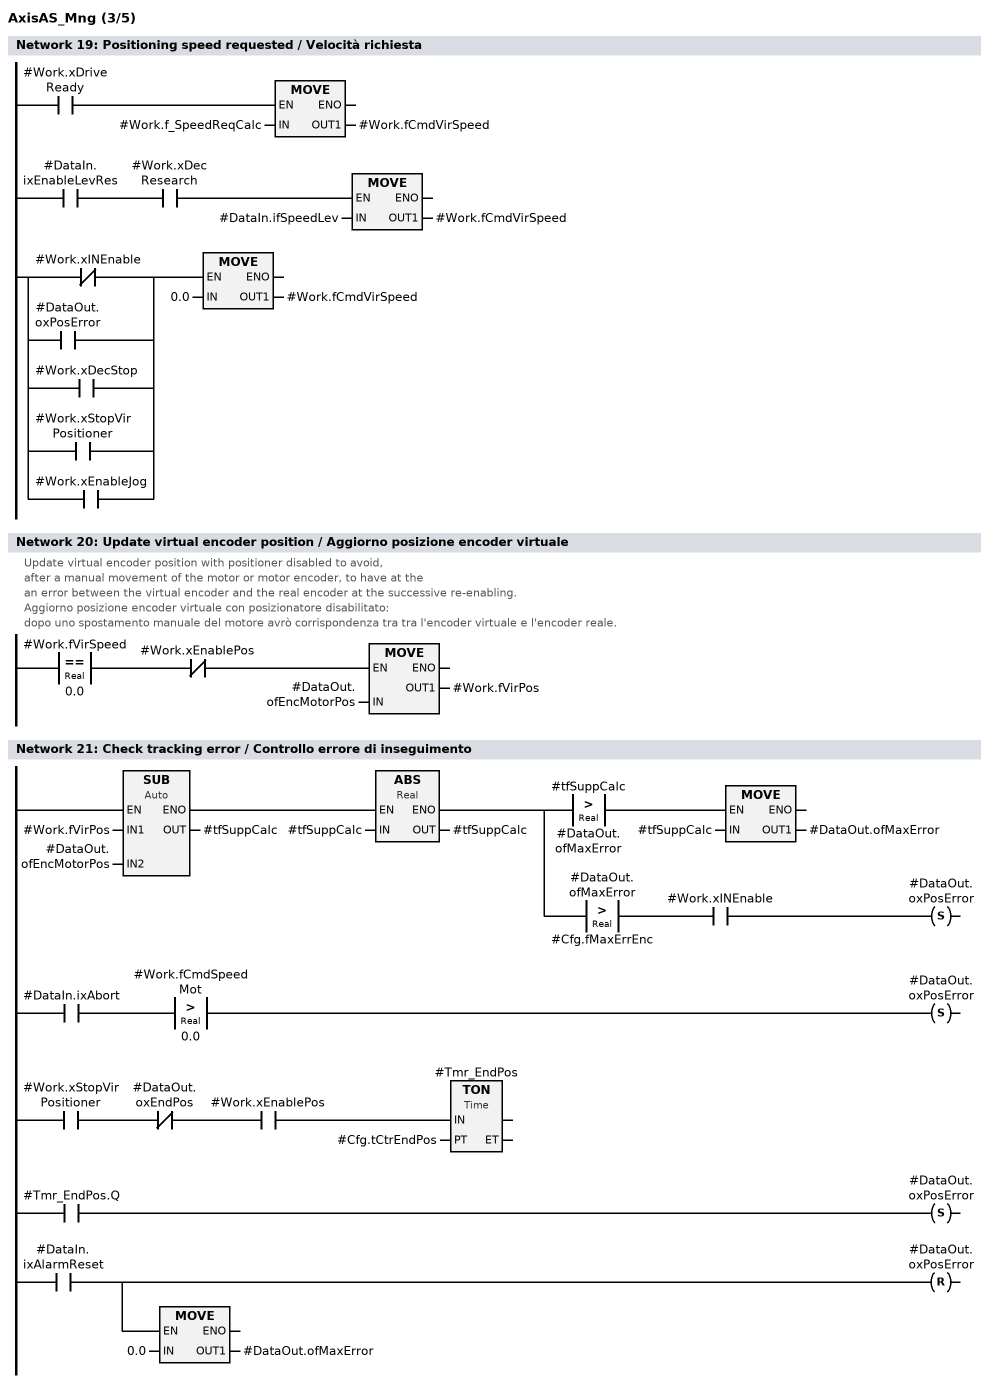
   RUNG wire#powerrail
      Contact( #Work.xDriveReady )
      Move(in := #Work.f_SpeedReqCalc, out1 => #Work.fCmdVirSpeed)
   END_RUNG
   RUNG wire#powerrail
      Contact( #DataIn.ixEnableLevRes )
      Contact( #Work.xDecResearch )
      Move(in := #DataIn.ifSpeedLev, out1 => #Work.fCmdVirSpeed)
   END_RUNG
   RUNG wire#powerrail
      I_Contact( #Work.xINEnable )
      wire#w1
      Move(in := 0.0, out1 => #Work.fCmdVirSpeed)
   END_RUNG
   RUNG wire#powerrail
      Contact( #DataOut.oxPosError )
   END_RUNG wire#w1
   RUNG wire#powerrail
      Contact( #Work.xDecStop )
   END_RUNG wire#w1
   RUNG wire#powerrail
      Contact( #Work.xStopVirPositioner )
   END_RUNG wire#w1
   RUNG wire#powerrail
      Contact( #Work.xEnableJog )
   END_RUNG wire#w1
   // the same network as SCL:
   IF #Work.xDriveReady THEN #Work.fCmdVirSpeed := #Work.f_SpeedReqCalc; END_IF;
   IF #DataIn.ixEnableLevRes AND #Work.xDecResearch THEN #Work.fCmdVirSpeed := #DataIn.ifSpeedLev; END_IF;
   IF NOT #Work.xINEnable OR #DataOut.oxPosError OR #Work.xDecStop OR #Work.xStopVirPositioner OR #Work.xEnableJog THEN
       #Work.fCmdVirSpeed := 0.0;
   END_IF;
END_REGION

REGION Network 20: Update virtual encoder position / Aggiorno posizione encoder virtuale
   // Update virtual encoder position with positioner disabled to avoid, 
   // after a manual movement of the motor or motor encoder, to have at the 
   // an error between the virtual encoder and the real encoder at the successive re-enabling.
   // Aggiorno posizione encoder virtuale con posizionatore disabilitato: 
   // dopo uno spostamento manuale del motore avrò corrispondenza tra tra l'encoder virtuale e l'encoder reale.
   RUNG wire#powerrail
      { S7_Templates := "SrcType := Real" } EQ_Contact(in1 := #Work.fVirSpeed, in2 := 0.0)
      I_Contact( #Work.xEnablePos )
      Move(in := #DataOut.ofEncMotorPos, out1 => #Work.fVirPos)
   END_RUNG
   // the same network as SCL:
   IF (#Work.fVirSpeed = 0.0) AND NOT #Work.xEnablePos THEN #Work.fVirPos := #DataOut.ofEncMotorPos; END_IF;
END_REGION

REGION Network 21: Check tracking error / Controllo errore di inseguimento
   RUNG wire#powerrail
      Sub(in1 := #Work.fVirPos, in2 := #DataOut.ofEncMotorPos, out => #tfSuppCalc)
      { S7_Templates := "SrcType := Real" } Abs(in := #tfSuppCalc, out => #tfSuppCalc)
      wire#w1
      { S7_Templates := "SrcType := Real" } GT_Contact(in1 := #tfSuppCalc, in2 := #DataOut.ofMaxError)
      Move(in := #tfSuppCalc, out1 => #DataOut.ofMaxError)
   END_RUNG
   RUNG wire#w1
      { S7_Templates := "SrcType := Real" } GT_Contact(in1 := #DataOut.ofMaxError, in2 := #Cfg.fMaxErrEnc)
      Contact( #Work.xINEnable )
      S_Coil( #DataOut.oxPosError )
   END_RUNG
   RUNG wire#powerrail
      Contact( #DataIn.ixAbort )
      { S7_Templates := "SrcType := Real" } GT_Contact(in1 := #Work.fCmdSpeedMot, in2 := 0.0)
      S_Coil( #DataOut.oxPosError )
   END_RUNG
   RUNG wire#powerrail
      Contact( #Work.xStopVirPositioner )
      I_Contact( #DataOut.oxEndPos )
      Contact( #Work.xEnablePos )
      { S7_Templates := "time_type := Time" } #Tmr_EndPos.TON(pt := #Cfg.tCtrEndPos, et =>)
   END_RUNG
   RUNG wire#powerrail
      Contact( #Tmr_EndPos.Q )
      S_Coil( #DataOut.oxPosError )
   END_RUNG
   RUNG wire#powerrail
      Contact( #DataIn.ixAlarmReset )
      wire#w2
      R_Coil( #DataOut.oxPosError )
   END_RUNG
   RUNG wire#w2
      Move(in := 0.0, out1 => #DataOut.ofMaxError)
   END_RUNG
   // the same network as SCL:
   #tfSuppCalc := #Work.fVirPos - #DataOut.ofEncMotorPos;
   #tfSuppCalc := ABS(#tfSuppCalc);
   IF #tfSuppCalc > #DataOut.ofMaxError THEN #DataOut.ofMaxError := #tfSuppCalc; END_IF;
   IF (#DataOut.ofMaxError > #Cfg.fMaxErrEnc) AND #Work.xINEnable THEN #DataOut.oxPosError := TRUE; END_IF;
   IF #DataIn.ixAbort AND (#Work.fCmdSpeedMot > 0.0) THEN #DataOut.oxPosError := TRUE; END_IF;
   #Tmr_EndPos.TON(IN := #Work.xStopVirPositioner AND NOT #DataOut.oxEndPos AND #Work.xEnablePos,
                   PT := #Cfg.tCtrEndPos);
   IF #Tmr_EndPos.Q THEN #DataOut.oxPosError := TRUE; END_IF;
   IF #DataIn.ixAlarmReset THEN
       #DataOut.oxPosError := FALSE;
       #DataOut.ofMaxError := 0.0;
   END_IF;
END_REGION

REGION Network 22 (SCL): Calcolo correzione PID

   #Work."fLim+Ppid" :=   (#Cfg.fMaxSpeed * 0.2);
   #Work."fLim-Ppid" := - (#Cfg.fMaxSpeed * 0.2);


   IF (#DataIn.ixEnableLevRes AND #Work.xDecResearch AND NOT #Work.xDecStop) OR #DataOut.oxEndPos THEN
       #Work.fMemoMaxSpeed := 1;
   END_IF;

   IF (ABS(#Work.fVirSpeed) > #Work.fMemoMaxSpeed) THEN
       #Work.fMemoMaxSpeed := #Work.fVirSpeed;
   END_IF;
   #Work.fSuppCalcPpid := ((#Work.fMemoMaxSpeed - #Work.fVirSpeed) / #Work.fMemoMaxSpeed) * #Cfg.fKPpidDec_Pos + #Cfg.fKPpid_Pos;
END_REGION

REGION Network 23 (SCL): Amplifico correzione PID a piramide su posizionamento
   #Work.fPpid := (#Work.fVirPos - #DataOut.ofEncMotorPos) * #Work.fSuppCalcPpid;
   IF #DataOut.oxCmdMotorBack THEN
       #Work.fPpid := - (#Work.fVirPos - #DataOut.ofEncMotorPos) * #Work.fSuppCalcPpid;
   END_IF;


   IF #Work.fPpid > #Work."fLim+Ppid" THEN
       #Work.fPpid := #Work."fLim+Ppid";
   END_IF;
   IF #Work.fPpid < #Work."fLim-Ppid" THEN
       #Work.fPpid := #Work."fLim-Ppid";
   END_IF;

   //Con posizionatore disabilitato azzero la parte proporzionale

   IF NOT #Work.xEnablePos OR #Work.xStopVirPositioner OR #DataOut.oxPosError THEN
       #Work.fPpid := 0;
   END_IF;

   // IF NOT #WORK.xEnablePos OR #WORK.xStopPositioner OR
   //     #WORK.fVirSpeed <= #CFG.fMinSpeed OR
   //     (NOT(#WORK.xINEnable) AND #WORK.fVirSpeed < 10) OR
   //     (ABS(#WORK.fNewPositionReq - #IN.ifEncoder) < #CFG.fMotWindPos) OR #OUT.oxPosError THEN
   //     #WORK.fPpid := 0;
   // END_IF;
END_REGION

REGION Network 24 (SCL): Speed load for motor from jog or positioner / Carico velocità per motore da jog o posizionatore
   //#Work.fCmdSpeedMot := 0.0;

   // IF #WORK.xEnablePos AND (ABS(#IN.ifEncoder - #WORK.fNewPositionReq) >= #CFG.fMotWindPos) THEN
   IF #Work.xEnablePos THEN
       IF (ABS(#DataIn.ifEncoder - #Work.f_PositionTarget) >= #Cfg.fMotWindPos) THEN
           IF #Work.fVirSpeed + #Work.fPpid <= 0 THEN
               #Work.fCmdSpeedMot := #Work.fVirSpeed / 2;
           ELSE
               #Work.fCmdSpeedMot := #Work.fVirSpeed + #Work.fPpid;
           END_IF;
       END_IF;
       IF NOT #DataOut.oxEndPos AND #Work.xDecStop AND (#Work.fVirSpeed = 0) AND #Work.xINEnable
           OR (ABS(#DataIn.ifEncoder - #Work.f_PositionTarget) >= #Cfg.fMotWindPos) AND (#Work.fCmdSpeedMot < #Cfg.fMinSpeed)
           AND #Work.xINEnable AND #Work.xDriveReady
       THEN
           #Work.fCmdSpeedMot := #Cfg.fMinSpeed;
       END_IF;
   ELSE
       #Work.fCmdSpeedMot := 0.0;
   END_IF;

   IF #Work.xEnableJog THEN
       #Work.fCmdSpeedMot := #Work.fJogSpeed;
   END_IF;
END_REGION

REGION Network 25 (SCL): Out motor speed / Out velocità motore
   IF #Work.fCmdSpeedMot > 0.0 AND NOT( #DataIn.ixAbort) THEN
       #DataOut.ofSpeedRequest := #Work.fCmdSpeedMot;
       IF #Work.fCmdSpeedMot < #Cfg.fMinSpeed AND NOT (#DataOut.oxPosError) THEN
           #DataOut.ofSpeedRequest := #Cfg.fMinSpeed;
       END_IF;
       IF #Work.fCmdSpeedMot > #Cfg.fMaxSpeed  THEN
           #DataOut.ofSpeedRequest := #Cfg.fMaxSpeed;
       END_IF;

   ELSE
       #DataOut.ofSpeedRequest := 0;
   END_IF;
END_REGION

REGION Network 26 (SCL): OUT Confirms positioning carried out (stop speed) / OUT Conferma posizionamento eseguito (velocità stop)
   IF #DataOut.ofSpeedRequest = 0 THEN
       #DataOut.oxStopSpeed := TRUE;
   ELSE
       #DataOut.oxStopSpeed := FALSE;
   END_IF;

   #DataOut.ofEncMotorPos := #DataIn.ifEncoder;
END_REGION

REGION Network 27: OUT Confirms positioning carried out (positioning ended) / OUT Conferma posizionamento eseguito (posizionamento terminato) + Camma posizione allargata
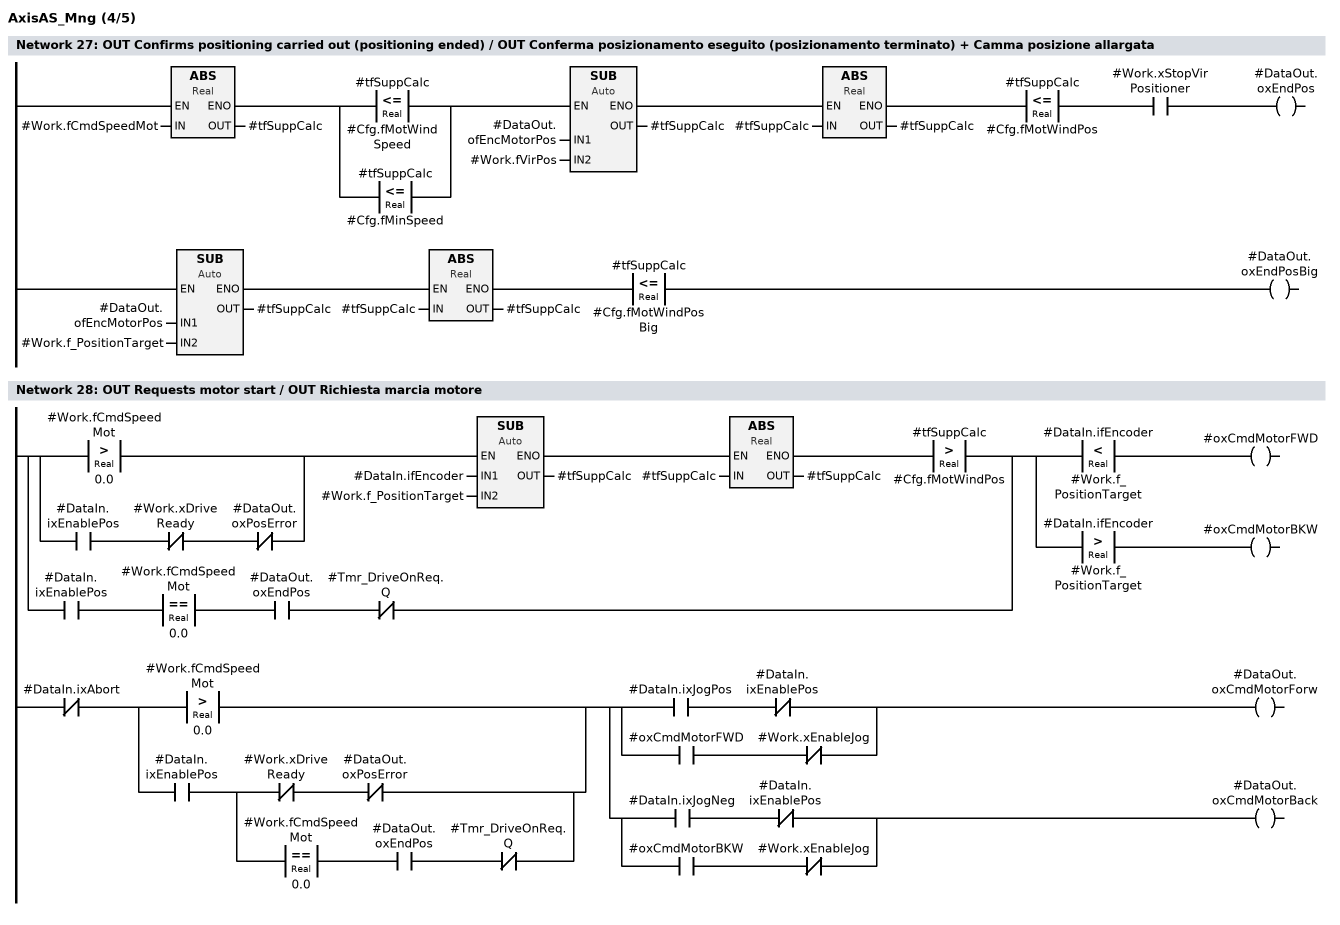
   RUNG wire#powerrail
      { S7_Templates := "SrcType := Real" } Abs(in := #Work.fCmdSpeedMot, out => #tfSuppCalc)
      wire#w1
      { S7_Templates := "SrcType := Real" } LE_Contact(in1 := #tfSuppCalc, in2 := #Cfg.fMotWindSpeed)
      wire#w2
      Sub(in1 := #DataOut.ofEncMotorPos, in2 := #Work.fVirPos, out => #tfSuppCalc)
      { S7_Templates := "SrcType := Real" } Abs(in := #tfSuppCalc, out => #tfSuppCalc)
      { S7_Templates := "SrcType := Real" } LE_Contact(in1 := #tfSuppCalc, in2 := #Cfg.fMotWindPos)
      Contact( #Work.xStopVirPositioner )
      Coil( #DataOut.oxEndPos )
   END_RUNG
   RUNG wire#w1
      { S7_Templates := "SrcType := Real" } LE_Contact(in1 := #tfSuppCalc, in2 := #Cfg.fMinSpeed)
   END_RUNG wire#w2
   RUNG wire#powerrail
      Sub(in1 := #DataOut.ofEncMotorPos, in2 := #Work.f_PositionTarget, out => #tfSuppCalc)
      { S7_Templates := "SrcType := Real" } Abs(in := #tfSuppCalc, out => #tfSuppCalc)
      { S7_Templates := "SrcType := Real" } LE_Contact(in1 := #tfSuppCalc, in2 := #Cfg.fMotWindPosBig)
      Coil( #DataOut.oxEndPosBig )
   END_RUNG
   // the same network as SCL:
   #tfSuppCalc := ABS(#Work.fCmdSpeedMot);
   #_w1 := (#tfSuppCalc <= #Cfg.fMotWindSpeed) OR (#tfSuppCalc <= #Cfg.fMinSpeed);
   IF #_w1 THEN
       #tfSuppCalc := #DataOut.ofEncMotorPos - #Work.fVirPos;
       #tfSuppCalc := ABS(#tfSuppCalc);
   END_IF;
   #DataOut.oxEndPos := #_w1 AND (#tfSuppCalc <= #Cfg.fMotWindPos) AND #Work.xStopVirPositioner;
   #tfSuppCalc := #DataOut.ofEncMotorPos - #Work.f_PositionTarget;
   #tfSuppCalc := ABS(#tfSuppCalc);
   #DataOut.oxEndPosBig := #tfSuppCalc <= #Cfg.fMotWindPosBig;
END_REGION

REGION Network 28: OUT Requests motor start / OUT Richiesta marcia motore
   RUNG wire#powerrail
      { S7_Templates := "SrcType := Real" } GT_Contact(in1 := #Work.fCmdSpeedMot, in2 := 0.0)
      wire#w1
      Sub(in1 := #DataIn.ifEncoder, in2 := #Work.f_PositionTarget, out => #tfSuppCalc)
      { S7_Templates := "SrcType := Real" } Abs(in := #tfSuppCalc, out => #tfSuppCalc)
      { S7_Templates := "SrcType := Real" } GT_Contact(in1 := #tfSuppCalc, in2 := #Cfg.fMotWindPos)
      wire#w2
      { S7_Templates := "SrcType := Real" } LT_Contact(in1 := #DataIn.ifEncoder, in2 := #Work.f_PositionTarget)
      Coil( #oxCmdMotorFWD )
   END_RUNG
   RUNG wire#powerrail
      Contact( #DataIn.ixEnablePos )
      I_Contact( #Work.xDriveReady )
      I_Contact( #DataOut.oxPosError )
   END_RUNG wire#w1
   RUNG wire#powerrail
      Contact( #DataIn.ixEnablePos )
      { S7_Templates := "SrcType := Real" } EQ_Contact(in1 := #Work.fCmdSpeedMot, in2 := 0.0)
      Contact( #DataOut.oxEndPos )
      I_Contact( #Tmr_DriveOnReq.Q )
   END_RUNG wire#w2
   RUNG wire#w2
      { S7_Templates := "SrcType := Real" } GT_Contact(in1 := #DataIn.ifEncoder, in2 := #Work.f_PositionTarget)
      Coil( #oxCmdMotorBKW )
   END_RUNG
   RUNG wire#powerrail
      I_Contact( #DataIn.ixAbort )
      wire#w3
      { S7_Templates := "SrcType := Real" } GT_Contact(in1 := #Work.fCmdSpeedMot, in2 := 0.0)
      wire#w4
      Contact( #DataIn.ixJogPos )
      I_Contact( #DataIn.ixEnablePos )
      wire#w6
      Coil( #DataOut.oxCmdMotorForw )
   END_RUNG
   RUNG wire#w3
      Contact( #DataIn.ixEnablePos )
      wire#w5
      I_Contact( #Work.xDriveReady )
      I_Contact( #DataOut.oxPosError )
   END_RUNG wire#w4
   RUNG wire#w5
      { S7_Templates := "SrcType := Real" } EQ_Contact(in1 := #Work.fCmdSpeedMot, in2 := 0.0)
      Contact( #DataOut.oxEndPos )
      I_Contact( #Tmr_DriveOnReq.Q )
   END_RUNG wire#w4
   RUNG wire#w4
      Contact( #oxCmdMotorFWD )
      I_Contact( #Work.xEnableJog )
   END_RUNG wire#w6
   RUNG wire#w4
      Contact( #DataIn.ixJogNeg )
      I_Contact( #DataIn.ixEnablePos )
      wire#w7
      Coil( #DataOut.oxCmdMotorBack )
   END_RUNG
   RUNG wire#w4
      Contact( #oxCmdMotorBKW )
      I_Contact( #Work.xEnableJog )
   END_RUNG wire#w7
   // the same network as SCL:
   #_w1 := (#Work.fCmdSpeedMot > 0.0) OR (#DataIn.ixEnablePos AND NOT #Work.xDriveReady AND NOT #DataOut.oxPosError);
   IF #_w1 THEN
       #tfSuppCalc := #DataIn.ifEncoder - #Work.f_PositionTarget;
       #tfSuppCalc := ABS(#tfSuppCalc);
   END_IF;
   #_w2 := (#_w1 AND (#tfSuppCalc > #Cfg.fMotWindPos)) OR (#DataIn.ixEnablePos AND (#Work.fCmdSpeedMot = 0.0) AND #DataOut.oxEndPos AND NOT #Tmr_DriveOnReq.Q);
   #oxCmdMotorFWD := #_w2 AND (#DataIn.ifEncoder < #Work.f_PositionTarget);
   #oxCmdMotorBKW := #_w2 AND (#DataIn.ifEncoder > #Work.f_PositionTarget);
   #_w3 := NOT #DataIn.ixAbort AND ((#Work.fCmdSpeedMot > 0.0) OR (#DataIn.ixEnablePos AND ((NOT #Work.xDriveReady AND NOT #DataOut.oxPosError) OR ((#Work.fCmdSpeedMot = 0.0) AND #DataOut.oxEndPos AND NOT #Tmr_DriveOnReq.Q))));
   #DataOut.oxCmdMotorForw := #_w3 AND ((#DataIn.ixJogPos AND NOT #DataIn.ixEnablePos) OR (#oxCmdMotorFWD AND NOT #Work.xEnableJog));
   #DataOut.oxCmdMotorBack := #_w3 AND ((#DataIn.ixJogNeg AND NOT #DataIn.ixEnablePos) OR (#oxCmdMotorBKW AND NOT #Work.xEnableJog));
END_REGION

REGION Network 29: OUT Requests motor start / OUT freno motore
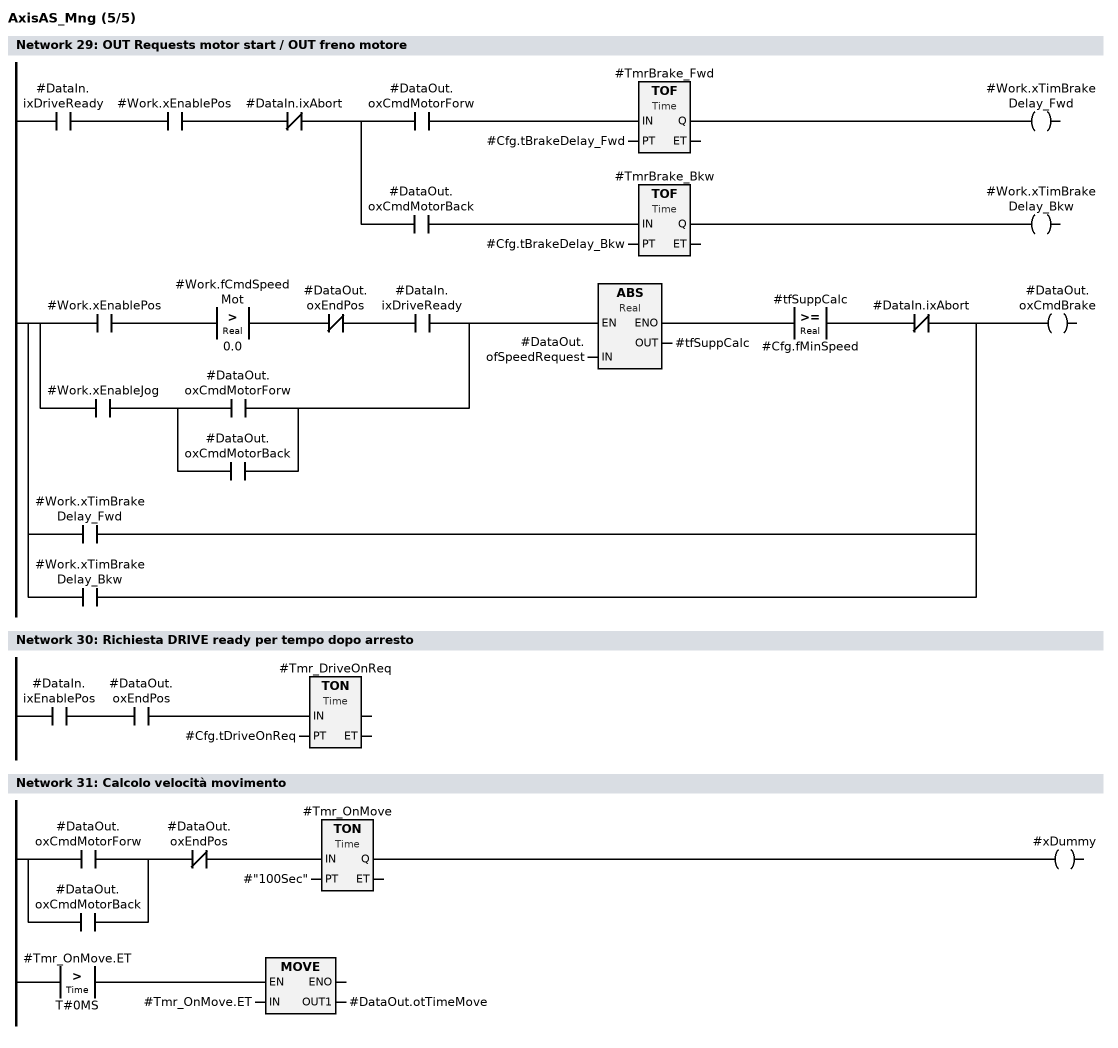
   RUNG wire#powerrail
      Contact( #DataIn.ixDriveReady )
      Contact( #Work.xEnablePos )
      I_Contact( #DataIn.ixAbort )
      wire#w1
      Contact( #DataOut.oxCmdMotorForw )
      { S7_Templates := "time_type := Time" } #TmrBrake_Fwd.TOF(pt := #Cfg.tBrakeDelay_Fwd, et =>)
      Coil( #Work.xTimBrakeDelay_Fwd )
   END_RUNG
   RUNG wire#w1
      Contact( #DataOut.oxCmdMotorBack )
      { S7_Templates := "time_type := Time" } #TmrBrake_Bkw.TOF(pt := #Cfg.tBrakeDelay_Bkw, et =>)
      Coil( #Work.xTimBrakeDelay_Bkw )
   END_RUNG
   RUNG wire#powerrail
      Contact( #Work.xEnablePos )
      { S7_Templates := "SrcType := Real" } GT_Contact(in1 := #Work.fCmdSpeedMot, in2 := 0.0)
      I_Contact( #DataOut.oxEndPos )
      Contact( #DataIn.ixDriveReady )
      wire#w2
      { S7_Templates := "SrcType := Real" } Abs(in := #DataOut.ofSpeedRequest, out => #tfSuppCalc)
      { S7_Templates := "SrcType := Real" } GE_Contact(in1 := #tfSuppCalc, in2 := #Cfg.fMinSpeed)
      I_Contact( #DataIn.ixAbort )
      wire#w4
      Coil( #DataOut.oxCmdBrake )
   END_RUNG
   RUNG wire#powerrail
      Contact( #Work.xEnableJog )
      wire#w3
      Contact( #DataOut.oxCmdMotorForw )
   END_RUNG wire#w2
   RUNG wire#w3
      Contact( #DataOut.oxCmdMotorBack )
   END_RUNG wire#w2
   RUNG wire#powerrail
      Contact( #Work.xTimBrakeDelay_Fwd )
   END_RUNG wire#w4
   RUNG wire#powerrail
      Contact( #Work.xTimBrakeDelay_Bkw )
   END_RUNG wire#w4
   // the same network as SCL:
   #_w1 := #DataIn.ixDriveReady AND #Work.xEnablePos AND NOT #DataIn.ixAbort;
   #TmrBrake_Fwd.TOF(IN := #_w1 AND #DataOut.oxCmdMotorForw, PT := #Cfg.tBrakeDelay_Fwd);
   #Work.xTimBrakeDelay_Fwd := #TmrBrake_Fwd.Q;
   #TmrBrake_Bkw.TOF(IN := #_w1 AND #DataOut.oxCmdMotorBack, PT := #Cfg.tBrakeDelay_Bkw);
   #Work.xTimBrakeDelay_Bkw := #TmrBrake_Bkw.Q;
   #_w2 := (#Work.xEnablePos AND (#Work.fCmdSpeedMot > 0.0) AND NOT #DataOut.oxEndPos AND #DataIn.ixDriveReady) OR (#Work.xEnableJog AND (#DataOut.oxCmdMotorForw OR #DataOut.oxCmdMotorBack));
   IF #_w2 THEN #tfSuppCalc := ABS(#DataOut.ofSpeedRequest); END_IF;
   #DataOut.oxCmdBrake := (#_w2 AND (#tfSuppCalc >= #Cfg.fMinSpeed) AND NOT #DataIn.ixAbort) OR #Work.xTimBrakeDelay_Fwd OR #Work.xTimBrakeDelay_Bkw;
END_REGION

REGION Network 30: Richiesta DRIVE ready per tempo dopo arresto
   RUNG wire#powerrail
      Contact( #DataIn.ixEnablePos )
      Contact( #DataOut.oxEndPos )
      { S7_Templates := "time_type := Time" } #Tmr_DriveOnReq.TON(pt := #Cfg.tDriveOnReq, et =>)
   END_RUNG
   // the same network as SCL:
   #Tmr_DriveOnReq.TON(IN := #DataIn.ixEnablePos AND #DataOut.oxEndPos, PT := #Cfg.tDriveOnReq);
END_REGION

REGION Network 31: Calcolo velocità movimento
   RUNG wire#powerrail
      Contact( #DataOut.oxCmdMotorForw )
      wire#w1
      I_Contact( #DataOut.oxEndPos )
      { S7_Templates := "time_type := Time" } #Tmr_OnMove.TON(pt := #"100Sec", et =>)
      Coil( #xDummy )
   END_RUNG
   RUNG wire#powerrail
      Contact( #DataOut.oxCmdMotorBack )
   END_RUNG wire#w1
   RUNG wire#powerrail
      { S7_Templates := "SrcType := Time" } GT_Contact(in1 := #Tmr_OnMove.ET, in2 := T#0MS)
      Move(in := #Tmr_OnMove.ET, out1 => #DataOut.otTimeMove)
   END_RUNG
   // the same network as SCL:
   #Tmr_OnMove.TON(IN := (#DataOut.oxCmdMotorForw OR #DataOut.oxCmdMotorBack) AND NOT #DataOut.oxEndPos,
                   PT := #"100Sec");
   #xDummy := #Tmr_OnMove.Q;
   IF #Tmr_OnMove.ET > T#0MS THEN #DataOut.otTimeMove := #Tmr_OnMove.ET; END_IF;
END_REGION
END_FUNCTION_BLOCK
